{attribute addProperty BoxType "EL3632-0000-0022"}
{attribute addProperty Id "StartTimeNextLatchAT %I*ULINT648"}
{attribute addProperty CRC "1335715474"}
{attribute addProperty SizeInBites "64"}
{attribute addProperty SizeInBytes "8"}
TYPE NextSync1Time_4F9D6692 :
STRUCT
	{attribute addProperty Name "StartTimeNextLatch"}
	StartTimeNextLatch AT %I* : ULINT;
END_STRUCT
END_TYPE

(* stored: Version 1.2.0.0, ProductVersion 3.1.4024.9
   DUT NextSync1Time_4F9D6692: Id {02e15d09-64e7-4c3d-b86c-88609b448a0e} *)
